TYPE ST_DefaultIdentityOUT3 :
STRUCT
	SKU						:STRING;
	GTIN					:STRING;
	ProductionOrder			:STRING;
	LocalProductionOrder	:STRING;
	PITCode					:STRING;
	BatchID					:STRING;
	ProductionLine			:STRING;
END_STRUCT
END_TYPE

(* stored: Version 1.1.0.1, ProductVersion 3.1.4024.13
   DUT ST_DefaultIdentityOUT3: Id {781092c9-20df-4062-8322-24a7c27c601e} *)
